// TIA Portal project "LAD_toggle_buttons" (V14)

(* hardware
DEVICE "S7-1200 station_1"  S7-1200 Station
   slot 0: "Rack_0"  S7-1200 Rack  Rack  V1.0
   slot 1: "PLC_1"  CPU 1214C AC/DC/Rly  6ES7 214-1BG40-0XB0  V4.2
*)

// ===== PLC "PLC_1"  CPU 1214C AC/DC/Rly =====

VAR_GLOBAL   // PLC tag table "Default tag table"
   "Call_button_1" AT %M2.0 : Bool;
   "Call_button_2" AT %M2.1 : Bool;
   "Call_button_3" AT %M2.2 : Bool;
   "Call_button_4" AT %M2.3 : Bool;
   "Call_button_5" AT %M2.4 : Bool;
   "S1_Out" AT %M2.5 : Bool;
   "S2_Out" AT %M2.6 : Bool;
   "S3_Out" AT %M2.7 : Bool;
   "S4_Out" AT %M3.0 : Bool;
   "S5_Out" AT %M3.1 : Bool;
   "Clear_button" AT %M3.2 : Bool;
END_VAR

DATA_BLOCK "Data_block_1"   // DB2
{ S7_Optimized_Access := 'TRUE' }
VERSION : 0.1
   VAR
      "Reset(SR_B1)" : Bool;
      "Triger(SR_B1)" : Bool;
      "Reset(SR_B2)" : Bool;
      "Reset(SR_B3)" : Bool;
      "Reset(SR_B4)" : Bool;
      "Reset(SR_B5)" : Bool;
      "Triger(SR_B2)" : Bool;
      "Triger(SR_B3)" : Bool;
      "Triger(SR_B4)" : Bool;
      "Triger(SR_B5)" : Bool;
   END_VAR
   VAR RETAIN
      max_signal_now : DInt;
      S1_in_queue : DInt;
      S2_in_queue : DInt;
      S3_in_queue : DInt;
      S4_in_queue : DInt;
      S5_in_queue : DInt;
   END_VAR
BEGIN
END_DATA_BLOCK

DATA_BLOCK "Block_1_DB"   // DB4
{ S7_Optimized_Access := 'TRUE' }
VERSION : 0.1
// stored: InstanceOfName Block_1
"Block_1"
BEGIN
END_DATA_BLOCK

// folder: System blocks/Program resources

DATA_BLOCK "IEC_Counter_0_DB"   // DB1
{ S7_Optimized_Access := 'TRUE' }
AUTHOR : Simatic
FAMILY : IEC
NAME : CNTR
VERSION : 1.0
// stored: InstanceOfName IEC_COUNTER
"IEC_COUNTER"
BEGIN
END_DATA_BLOCK

DATA_BLOCK "Big_State_Counter"   // DB3
{ S7_Optimized_Access := 'TRUE' }
AUTHOR : SIMATIC
FAMILY : IEC
NAME : DCNTR
VERSION : 1.2
// stored: InstanceOfName IEC_DCOUNTER
"IEC_DCOUNTER"
BEGIN
END_DATA_BLOCK

DATA_BLOCK "Button2"   // DB5
{ S7_Optimized_Access := 'TRUE' }
AUTHOR : Simatic
FAMILY : IEC
NAME : CNTR
VERSION : 1.0
// stored: InstanceOfName IEC_COUNTER
"IEC_COUNTER"
BEGIN
END_DATA_BLOCK

DATA_BLOCK "Button3"   // DB6
{ S7_Optimized_Access := 'TRUE' }
AUTHOR : Simatic
FAMILY : IEC
NAME : CNTR
VERSION : 1.0
// stored: InstanceOfName IEC_COUNTER
"IEC_COUNTER"
BEGIN
END_DATA_BLOCK

DATA_BLOCK "Button4"   // DB7
{ S7_Optimized_Access := 'TRUE' }
AUTHOR : Simatic
FAMILY : IEC
NAME : CNTR
VERSION : 1.0
// stored: InstanceOfName IEC_COUNTER
"IEC_COUNTER"
BEGIN
END_DATA_BLOCK

DATA_BLOCK "Button5"   // DB8
{ S7_Optimized_Access := 'TRUE' }
AUTHOR : Simatic
FAMILY : IEC
NAME : CNTR
VERSION : 1.0
// stored: InstanceOfName IEC_COUNTER
"IEC_COUNTER"
BEGIN
END_DATA_BLOCK

// folder: (top level)

FUNCTION_BLOCK "Block_1"   // FB1, LAD
{ S7_Optimized_Access := 'TRUE' }
VERSION : 0.1
   VAR_TEMP
      First_signal : DInt;
      cv : Int;
      cv2 : Int;
      cv3 : Int;
      cv4 : Int;
      cv5 : Int;
      last_signal_now : DInt;
      Big_State_Counter_Reset : Bool;
   END_VAR
   VAR_TEMP   // added for the SCL form of the ladder/FBD networks
      _w1 : Bool;
   END_VAR
BEGIN

REGION Network 1: Making ON-OFF for buttons, preventing "0" number in button-queue
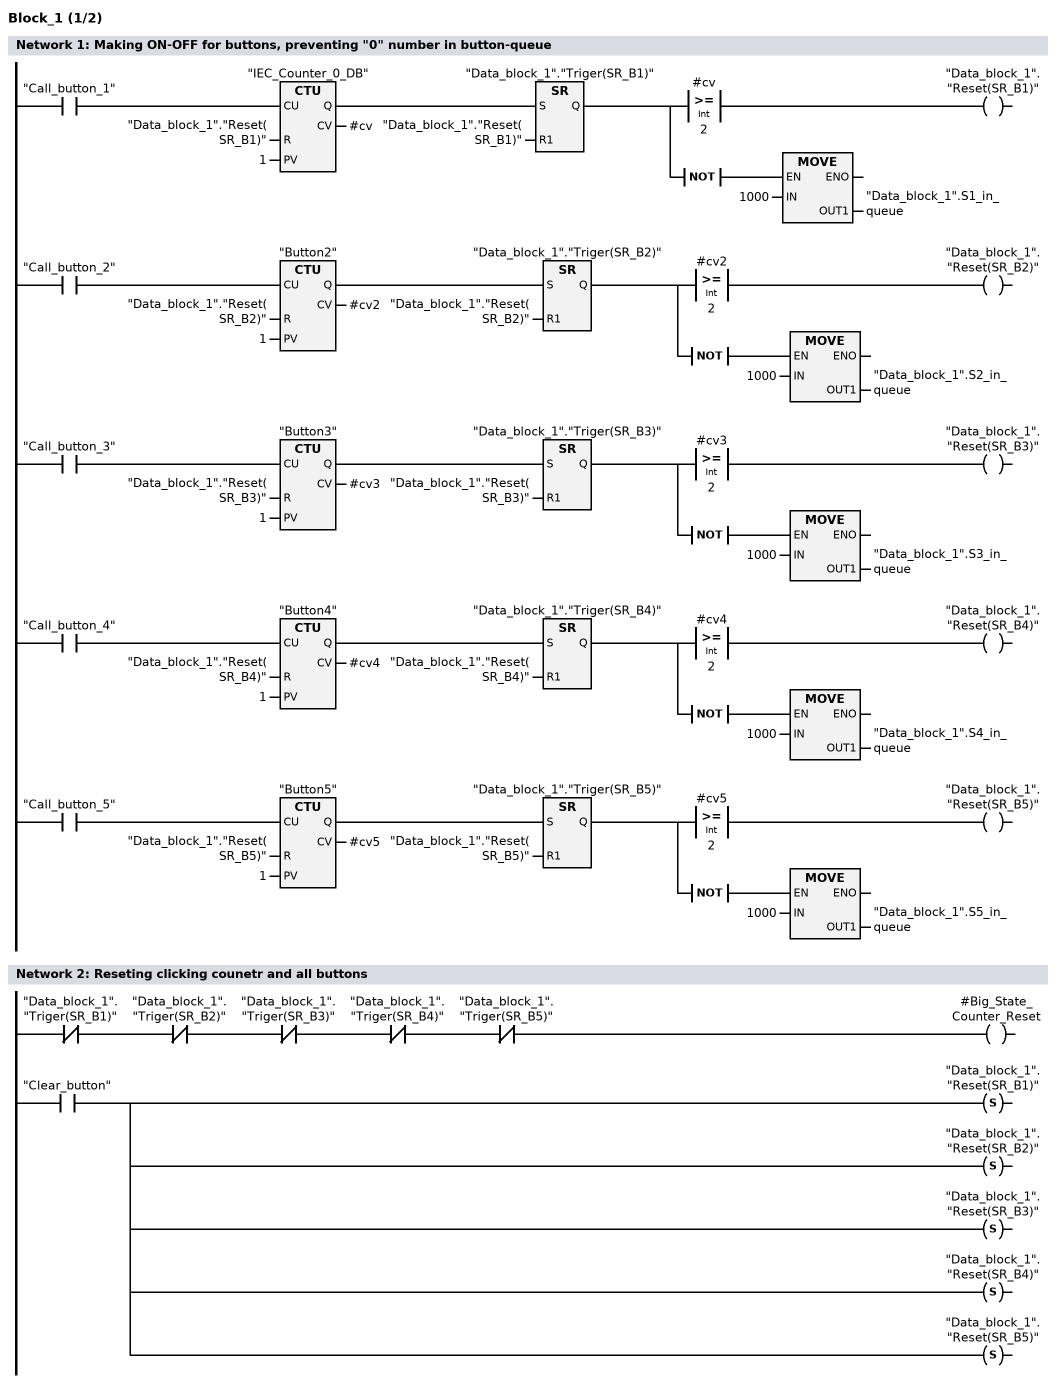
   "IEC_Counter_0_DB".CTU(CU := "Call_button_1", R := "Data_block_1"."Reset(SR_B1)", PV := 1, CV => #cv);
   IF "IEC_Counter_0_DB".Q THEN
       "Data_block_1"."Triger(SR_B1)" := TRUE;   // SR flip-flop
   END_IF;
   IF "Data_block_1"."Reset(SR_B1)" THEN "Data_block_1"."Triger(SR_B1)" := FALSE; END_IF;
   "Data_block_1"."Reset(SR_B1)" := "Data_block_1"."Triger(SR_B1)" AND (#cv >= 2);
   IF NOT "Data_block_1"."Triger(SR_B1)" THEN "Data_block_1".S1_in_queue := 1000; END_IF;
   "Button2".CTU(CU := "Call_button_2", R := "Data_block_1"."Reset(SR_B2)", PV := 1, CV => #cv2);
   IF "Button2".Q THEN
       "Data_block_1"."Triger(SR_B2)" := TRUE;   // SR flip-flop
   END_IF;
   IF "Data_block_1"."Reset(SR_B2)" THEN "Data_block_1"."Triger(SR_B2)" := FALSE; END_IF;
   "Data_block_1"."Reset(SR_B2)" := "Data_block_1"."Triger(SR_B2)" AND (#cv2 >= 2);
   IF NOT "Data_block_1"."Triger(SR_B2)" THEN "Data_block_1".S2_in_queue := 1000; END_IF;
   "Button3".CTU(CU := "Call_button_3", R := "Data_block_1"."Reset(SR_B3)", PV := 1, CV => #cv3);
   IF "Button3".Q THEN
       "Data_block_1"."Triger(SR_B3)" := TRUE;   // SR flip-flop
   END_IF;
   IF "Data_block_1"."Reset(SR_B3)" THEN "Data_block_1"."Triger(SR_B3)" := FALSE; END_IF;
   "Data_block_1"."Reset(SR_B3)" := "Data_block_1"."Triger(SR_B3)" AND (#cv3 >= 2);
   IF NOT "Data_block_1"."Triger(SR_B3)" THEN "Data_block_1".S3_in_queue := 1000; END_IF;
   "Button4".CTU(CU := "Call_button_4", R := "Data_block_1"."Reset(SR_B4)", PV := 1, CV => #cv4);
   IF "Button4".Q THEN
       "Data_block_1"."Triger(SR_B4)" := TRUE;   // SR flip-flop
   END_IF;
   IF "Data_block_1"."Reset(SR_B4)" THEN "Data_block_1"."Triger(SR_B4)" := FALSE; END_IF;
   "Data_block_1"."Reset(SR_B4)" := "Data_block_1"."Triger(SR_B4)" AND (#cv4 >= 2);
   IF NOT "Data_block_1"."Triger(SR_B4)" THEN "Data_block_1".S4_in_queue := 1000; END_IF;
   "Button5".CTU(CU := "Call_button_5", R := "Data_block_1"."Reset(SR_B5)", PV := 1, CV => #cv5);
   IF "Button5".Q THEN
       "Data_block_1"."Triger(SR_B5)" := TRUE;   // SR flip-flop
   END_IF;
   IF "Data_block_1"."Reset(SR_B5)" THEN "Data_block_1"."Triger(SR_B5)" := FALSE; END_IF;
   "Data_block_1"."Reset(SR_B5)" := "Data_block_1"."Triger(SR_B5)" AND (#cv5 >= 2);
   IF NOT "Data_block_1"."Triger(SR_B5)" THEN "Data_block_1".S5_in_queue := 1000; END_IF;
END_REGION

REGION Network 2: Reseting clicking counetr and all buttons
   RUNG wire#powerrail
      I_Contact( "Data_block_1"."Triger(SR_B1)" )
      I_Contact( "Data_block_1"."Triger(SR_B2)" )
      I_Contact( "Data_block_1"."Triger(SR_B3)" )
      I_Contact( "Data_block_1"."Triger(SR_B4)" )
      I_Contact( "Data_block_1"."Triger(SR_B5)" )
      Coil( #Big_State_Counter_Reset )
   END_RUNG
   RUNG wire#powerrail
      Contact( "Clear_button" )
      wire#w1
      S_Coil( "Data_block_1"."Reset(SR_B1)" )
   END_RUNG
   RUNG wire#w1
      S_Coil( "Data_block_1"."Reset(SR_B2)" )
   END_RUNG
   RUNG wire#w1
      S_Coil( "Data_block_1"."Reset(SR_B3)" )
   END_RUNG
   RUNG wire#w1
      S_Coil( "Data_block_1"."Reset(SR_B4)" )
   END_RUNG
   RUNG wire#w1
      S_Coil( "Data_block_1"."Reset(SR_B5)" )
   END_RUNG
   // the same network as SCL:
   #Big_State_Counter_Reset := NOT "Data_block_1"."Triger(SR_B1)" AND NOT "Data_block_1"."Triger(SR_B2)" AND NOT "Data_block_1"."Triger(SR_B3)" AND NOT "Data_block_1"."Triger(SR_B4)" AND NOT "Data_block_1"."Triger(SR_B5)";
   IF "Clear_button" THEN
       "Data_block_1"."Reset(SR_B1)" := TRUE;
       "Data_block_1"."Reset(SR_B2)" := TRUE;
       "Data_block_1"."Reset(SR_B3)" := TRUE;
       "Data_block_1"."Reset(SR_B4)" := TRUE;
       "Data_block_1"."Reset(SR_B5)" := TRUE;
   END_IF;
END_REGION

REGION Network 3: Making button-queue
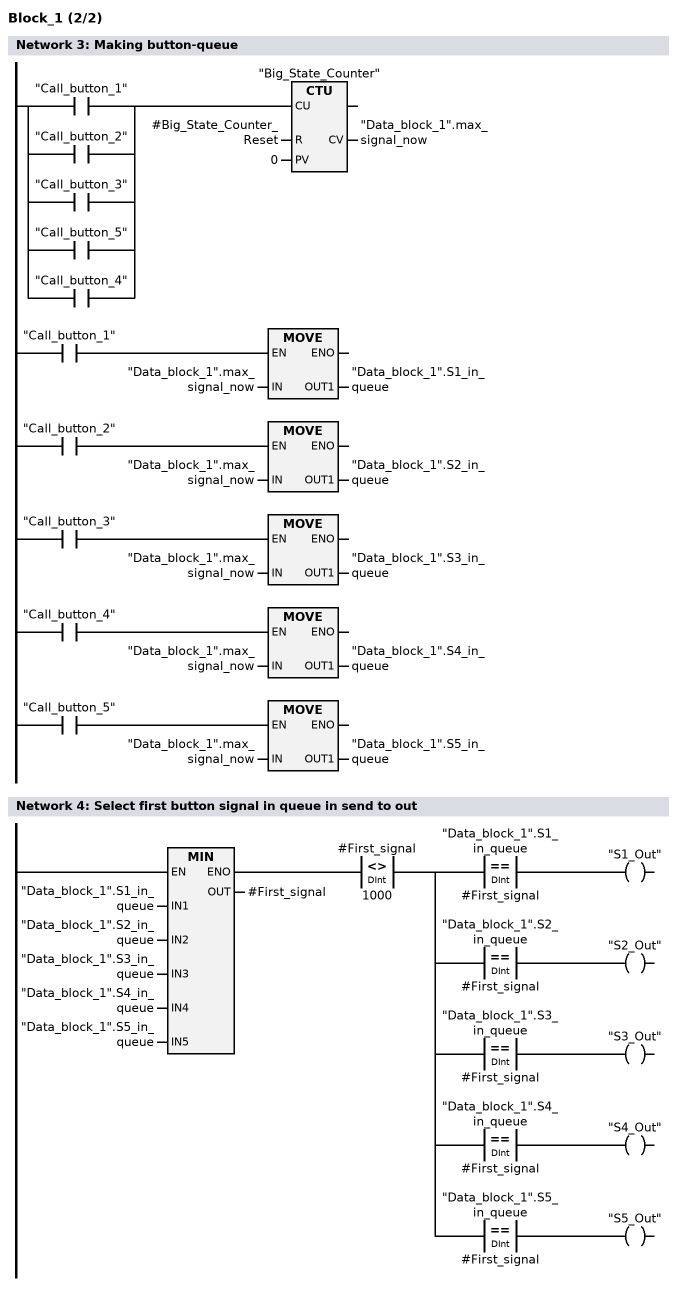
   "Big_State_Counter".CTU(CU := "Call_button_1" OR "Call_button_2" OR "Call_button_3" OR "Call_button_5" OR "Call_button_4",
                           R := #Big_State_Counter_Reset,
                           PV := 0,
                           CV => "Data_block_1".max_signal_now);
   IF "Call_button_1" THEN "Data_block_1".S1_in_queue := "Data_block_1".max_signal_now; END_IF;
   IF "Call_button_2" THEN "Data_block_1".S2_in_queue := "Data_block_1".max_signal_now; END_IF;
   IF "Call_button_3" THEN "Data_block_1".S3_in_queue := "Data_block_1".max_signal_now; END_IF;
   IF "Call_button_4" THEN "Data_block_1".S4_in_queue := "Data_block_1".max_signal_now; END_IF;
   IF "Call_button_5" THEN "Data_block_1".S5_in_queue := "Data_block_1".max_signal_now; END_IF;
END_REGION

REGION Network 4: Select first button signal in queue in send to out
   #First_signal := MIN(IN1 := "Data_block_1".S1_in_queue, IN2 := "Data_block_1".S2_in_queue, IN3 := "Data_block_1".S3_in_queue, IN4 := "Data_block_1".S4_in_queue, IN5 := "Data_block_1".S5_in_queue);
   #_w1 := #First_signal <> 1000;
   "S1_Out" := #_w1 AND ("Data_block_1".S1_in_queue = #First_signal);
   "S2_Out" := #_w1 AND ("Data_block_1".S2_in_queue = #First_signal);
   "S3_Out" := #_w1 AND ("Data_block_1".S3_in_queue = #First_signal);
   "S4_Out" := #_w1 AND ("Data_block_1".S4_in_queue = #First_signal);
   "S5_Out" := #_w1 AND ("Data_block_1".S5_in_queue = #First_signal);
END_REGION
END_FUNCTION_BLOCK

ORGANIZATION_BLOCK "Main"   // OB1, LAD, ProgramCycle
TITLE = "Main Program Sweep (Cycle)"
{ S7_Optimized_Access := 'TRUE' }
VERSION : 0.1
   VAR_INPUT
      Initial_Call : Bool;   // Initial call of this OB
      Remanence : Bool;   // =True, if remanent data are available
   END_VAR
BEGIN

REGION Network 1
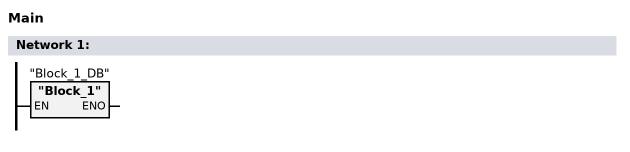
   RUNG wire#powerrail
      "Block_1_DB"()
   END_RUNG
   // the same network as SCL:
   "Block_1_DB"();   // "Block_1"
END_REGION
END_ORGANIZATION_BLOCK